// SIMATIC S7-200 project (STEP 7-Micro/WIN), CPU 226 REL 02.01

ORGANIZATION_BLOCK OB_1:OB1
TITLE=PROGRAM COMMENTS
// 食品或饮料行业的自动灌装机06 系统，通过启动灌装机，并在饮料瓶装生产线上精确控制瓶子的定位、灌装和封盖流程。
// 操作员按下启动按钮启动系统，设备通过上管控制将包装管送入位置，随后压板控制和压管控制分别在不同阶段固定管材。灌装阀和注料控制接着在各自脉冲范围内开始灌装液体。为了确保灌装一致性，注料控制和灌装阀应在编码器脉冲计数器的相同脉冲范围内动作，但目前两者的脉冲范围略有差异。运行状态指示灯在无故障信号A和故障信号B时点亮，显示设备运行，而启动按钮的信号通过其他逻辑参与控制。若故障信号A或故障信号B触发，例如电机故障或压力异常，运行状态指示灯立即熄灭。
// 系统通过编码器脉冲计数器精确记录灌装位置，色标传感器检测包装上的色标，确保灌装对准。灌装过程中，加热控制维持液体温度，但只有在冷却控制和风机控制均开启时才会激活，以避免温度失控。冷却控制、风机控制、搅拌控制和保温控制分别工作以维持灌装环境稳定，例如保持化妆品乳液的适宜粘度。若温度传感器检测到异常，系统暂停灌装并调整环境。压管传感器检测压管是否到位，置位压管到位标志，触发后续动作。
// 急停按钮被按下时，所有动作输出如上管控制、灌装阀、压板控制等应立即停止，但当前仅部分标志复位，需进一步完善。
BEGIN
Network 1
// 初始一次 on 系统初始化
LD     SM0.0
CALL   SBR_9:SBR9
?000
Network 2 // Network Title
// 运行初始化 （数据显示）
LD     SM0.1
CALL   SBR_0:SBR0
CALL   SBR_3:SBR3
=      M5.1
MOVW   +0, VW30
S      M1.1, 1
Network 3
// 恢复参数出厂设置
LD     M0.3
CALL   SBR_1:SBR1
Network 4
// 保存参数
LD     M0.4
CALL   SBR_2:SBR2
Network 5
// 参数修改后，未确定保存，参数恢复正常
LD     M2.4
CALL   SBR_3:SBR3
Network 6
// 大盘正常运行
LD     I1.2
O      M6.3
A      I0.5
AN     Q0.1
=      M6.3
EU
MOVW   +0, VW30
Network 7
// 点动运行
LD     I1.3
AN     Q0.1
=      M6.2
Network 8
LD     SM0.1
S      M2.0, 1
Network 9
// 大盘运行
LD     M6.2
O      M6.3
AN     Q0.1
EU
S      M20.6, 1
Network 10
// 点动停止
LD     M6.2
ED
R      M20.6, 1
Network 11
// 运行停机
LDD>=  HC0, +2300
AD<=   HC0, +2350
AN     M6.2
AN     M6.3
EU
R      M20.6, 1
Network 12
// 生产速度，计数设定，产量计数的BCD转换
LD     SM0.0
MOVW   VW10, VW54
BCDI   VW54
MOVW   VW14, VW50
BCDI   VW50
MOVW   VW52, VW18
IBCD   VW18
Network 13
// 手动升降速，及速度限制（速度必须在10-90之间)
LD     M1.1
LPS
AW>    VW54, +91
MOVW   +90, VW54
MOVW   VW54, VW10
IBCD   VW10
LRD
AW<    VW54, +10
MOVW   +10, VW54
MOVW   VW54, VW10
IBCD   VW10
LRD
AW<    VW54, +91
A      SM0.5
EU
A      M2.1
+I     +1, VW54
MOVW   VW54, VW10
IBCD   VW10
LPP
AW>    VW54, +10
A      SM0.5
EU
A      M2.2
-I     +1, VW54
MOVW   VW54, VW10
IBCD   VW10
Network 14
// 转速换算，根据大盘速度换算电机转速
LD     M1.1
MOVW   VW54, LW2
AENO
MUL    +44, LD0
AENO
MOVD   LD0, VD480
AENO
/D     +47, VD480
AENO
DTR    VD480, VD504
Network 15
// 真空 
LD     M1.1
A      M10.0
AN     M2.0
AN     Q0.1
=      Q0.7
Network 16
// 压板
LD     M1.1
AW>=   VW30, +2
A      M10.2
AN     M2.0
AN     M4.2
AD>=   HC0, VD140
AD<=   HC0, VD128
=      Q1.2
Network 17
// 上管
LD     M1.1
AW>=   VW30, +2
A      M2.7
AN     M2.0
AD>=   HC0, VD100
AD<=   HC0, +200
AN     M4.2
EU
S      Q0.2, 1
Network 18
// 上管回
LDD>=  HC0, +1150
ON     I0.5
EU
R      Q0.2, 1
Network 19
// 拨管
LD     M1.1
A      M10.2
AN     M2.0
AN     M4.2
=      Q1.3
Network 20
// 压管下
LD     M1.0
AW>=   VW30, +2
LD     M1.1
A      M10.1
OLD
AD>=   HC0, +1100
EU
S      Q1.7, 1
Network 21
// 净化，洗尘
LD     M3.0
A      M1.1
AD>=   HC0, VD104
AD<=   HC0, VD304
AN     M2.0
=      Q0.3
Network 22
// 停机复位 Q2.3未用 Q1.2压板 Q1.7压管 Q1.1灌装阀
LDN    M20.6
O      Q0.1
S      Q2.3, 1
R      Q1.2, 1
R      Q1.7, 1
EU
R      Q1.1, 1
Network 23
// 压管回
LD     I1.5
EU
R      Q1.7, 1
Network 24
// 允许脉冲输出,步进电机转动进行色标检测. M29.6状态取反（复位表示置位）
LDD>=  HC0, +1000
AD<=   HC0, +1050
EU
R      M29.6, 1
Network 25
// 禁止进行色标检测 M29.6状态取反（置位表示复位）
LDD>=  HC0, +1800
AD<=   HC0, +1850
EU
S      M29.6, 1
Network 26
// 色标电机停止转动 表示同步电机机械定位分开脱离停止旋转（上升结合旋转）
LDD>=  HC0, +2000
AD<=   HC0, +2050
MOVB   16#5, SMB67
PLS    0
Network 27
// 找到色标,步进停止转动
LD     I0.3
A      M20.5
LDN    I0.3
AN     M20.5
OLD
EU
MOVB   16#5, SMB67
PLS    0
Network 28
// 色标检测脉冲输出
LD     M1.1
A      M3.1
LDN    M25.0
A      I0.3
LD     M25.0
AN     I0.3
OLD
ALD
AN     M29.6
EU
AN     Q0.1
MOVB   16#85, SMB67
MOVW   +860, SMW68
MOVD   +99999999, SMD72
PLS    0
Network 29
// 检管信号记忆，注料启动
LDN    M2.0
ANI    I0.6
EU
S      M4.0, 1
Network 30
// 料塞
LD     M3.2
A      M1.1
AD>=   HC0, VD124
AD<=   HC0, VD132
AN     M2.0
A      M5.0
=      Q1.1
Network 31
// 注料
LD     M3.2
A      M1.1
AD>=   HC0, VD108
AD<=   HC0, VD112
AN     M2.0
A      M5.0
=      Q0.4
Network 32
// 吹气，并复位检管信号
LD     M3.2
A      M1.1
AD>=   HC0, VD116
AD<=   HC0, VD120
AN     M2.0
A      M5.0
=      Q0.5
Network 33
// 加热（必须先打开冷却，和风机才能正常工作）
LD     M1.0
O      M1.1
A      M10.4
A      Q1.6
A      Q1.5
=      Q1.4
NOT
R      M10.4, 1
Network 34
// 冷却
LD     M1.1
A      M10.3
O      Q1.5
=      Q1.5
Network 35
// 关闭冷却
LD     M10.3
ED
LPS
AN     M10.4
R      Q1.5, 1
LPP
A      M10.4
S      M10.3, 1
Network 36
// 风机
LD     M1.1
A      M3.3
O      Q1.6
=      Q1.6
Network 37
// 关闭风机
LD     M3.3
ED
LPS
AN     M10.4
R      Q1.6, 1
LPP
A      M10.4
S      M3.3, 1
Network 38
// 搅拌
LD     M1.1
A      M3.5
=      Q0.6
Network 39
// 保温
LD     M1.1
A      M3.6
=      Q1.0
Network 40
// 大盘运行停止,上管压管终止
LDN    M6.3
EU
R      M2.7, 1
R      M10.1, 2
Network 41
// 计数到标志位
LD     M1.4
AW>=   VW52, VW50
=      M4.2
Network 42
// 记数
LD     M1.1
AW<    VW52, VW50
A      Q0.4
EU
A      M1.4
INCW   VW52
Network 43
// 计数清零
LD     M1.3
MOVW   +0, VW52
Network 44
// 故障时，复位脉冲输出停机
LD     Q0.1
EU
R      M20.6, 1
MOVB   16#5, SMB67
PLS    0
Network 45
// USS协议
LD     SM0.0
=      L60.0
LD     M20.6
=      L63.7
LD     SM0.1
=      L63.6
LD     SM0.1
=      L63.5
LD     SM0.1
=      L63.4
LDN    SM0.0
=      L63.3
LD     L60.0
CALL   USS_CTRL:SBR8, L63.7, L63.6, L63.5, L63.4, L63.3, 1, 1, VD504, V500.3, VB514, VW516, VD510, V500.4, V500.5, V500.6, V500.7
Network 46
// 故障输出
LDN    I0.7
ON     I1.0
O      M13.0
=      Q0.1
Network 47
// 故障分类，触摸屏显示故障信息
LD     SM0.0
LPS
AN     I0.7
=      M20.0
LRD
AN     I1.0
=      M20.1
LPP
A      M13.0
=      M20.3
Network 48
// A门B门手盘车
LD     SM0.0
LPS
AN     I1.6
=      M13.1
LRD
AN     I1.7
=      M13.2
LPP
AN     I2.1
=      M13.3
Network 49
// 故障汇总
LD     M13.1
O      M13.3
O      M13.2
=      M13.0
Network 50
// 故障报警弹画面
LD     SM0.0
LPS
A      Q0.1
MOVW   +17, VW254
LPP
AN     Q0.1
EU
MOVW   +12, VW254
Network 51
// 画面值进行BCD转换
LD     SM0.0
MOVW   VW254, VW256
IBCD   VW256
Network 52
LD     SM0.0
DTI    HC0, VW180
MOVW   VW180, VW184
IBCD   VW184
END_ORGANIZATION_BLOCK

SUBROUTINE_BLOCK SBR_0:SBR0
TITLE=SUBROUTINE COMMENTS
BEGIN
Network 1 // Network Title
// Network Comment 开机时，所有数据清零
LD     SM0.0
R      Q0.0, 24
R      M0.0, 100
R      M10.0, 6
R      M25.0, 1
MOVD   +2330, VD1012
Network 2
// 高速计数器（编码器定义）
LD     SM0.0
MOVB   16#F8, SMB37
HDEF   0, 10
MOVD   +0, SMD38
MOVD   +30000, SMD42
ATCH   INT_0:INT0, 28
ENI
HSC    0
Network 3
// 步进电机脉冲定义（16#85为脉冲时间定义） SMD67脉冲参数 SMD68脉冲周期 SMD72脉冲数 (ATCH为中断控制  其中 INT_4 控制色标 7 为下降沿脉冲， 6 为上升沿脉冲)
LD     SM0.0
LPS
MOVB   16#85, SMB67
MOVW   +900, SMW68
MOVD   +99999999, SMD72
AN     M25.0
ATCH   INT_4:INT4, 7
LRD
A      M25.0
ATCH   INT_4:INT4, 6
LPP
ENI
Network 4
// 下列表示变频器与PLC之间通讯协议，1为模式 ，19200 为通讯速率， 16#02 为变频器地址 ， v500.0为变频器状态反馈地址（回答）
//  vb514为故障反馈地址
LD     SM0.0
CALL   USS_INIT:SBR5, 1, 19200, 16#2, V500.0, VB514
END_SUBROUTINE_BLOCK

SUBROUTINE_BLOCK SBR_1:SBR1
TITLE=
BEGIN
Network 1
// 机器工位编码器的脉冲位置（初始化时，将下列各值强制输入到设备内部）
LD     SM0.0
MOVW   +50, VW200
MOVW   +700, VW1004
MOVW   +800, VW208
MOVW   +1700, VW212
MOVW   +2000, VW216
MOVW   +2100, VW220
MOVW   +780, VW224
MOVW   +800, VW228
MOVW   +1600, VW232
MOVW   +2000, VW236
MOVW   +300, VW240
MOVW   +1800, VW150
Network 2
// 工位脉冲数值转换触摸屏代码显示
LD     SM0.0
MOVW   VW200, VW400
IBCD   VW400
MOVW   VW1004, VW404
IBCD   VW404
MOVW   VW208, VW408
IBCD   VW408
MOVW   VW212, VW412
IBCD   VW412
MOVW   VW216, VW416
IBCD   VW416
MOVW   VW220, VW420
IBCD   VW420
MOVW   VW224, VW424
IBCD   VW424
MOVW   VW228, VW428
IBCD   VW428
MOVW   VW232, VW432
IBCD   VW432
MOVW   VW236, VW436
IBCD   VW436
MOVW   VW240, VW440
IBCD   VW440
MOVW   VW150, VW152
IBCD   VW152
END_SUBROUTINE_BLOCK

SUBROUTINE_BLOCK SBR_2:SBR2
TITLE=
BEGIN
Network 1
// 确定数据保存（数据修改后确认）触摸屏及plc数据转换
LD     SM0.0
MOVW   VW400, VW200
BCDI   VW200
MOVW   VW404, VW1004
BCDI   VW1004
MOVW   VW408, VW208
BCDI   VW208
MOVW   VW412, VW212
BCDI   VW212
MOVW   VW416, VW216
BCDI   VW216
MOVW   VW420, VW220
BCDI   VW220
MOVW   VW424, VW224
BCDI   VW224
MOVW   VW428, VW228
BCDI   VW228
MOVW   VW432, VW232
BCDI   VW232
MOVW   VW436, VW236
BCDI   VW236
MOVW   VW440, VW240
BCDI   VW240
MOVW   VW152, VW150
BCDI   VW150
Network 2
LD     SM0.0
ITD    VW200, VD100
ITD    VW1004, VD104
ITD    VW208, VD108
ITD    VW212, VD112
ITD    VW216, VD116
ITD    VW220, VD120
ITD    VW224, VD124
ITD    VW228, VD128
ITD    VW232, VD132
ITD    VW236, VD136
ITD    VW240, VD140
ITD    VW150, VD160
Network 3
LD     SM0.0
MOVD   VD104, VD304
+D     +320, VD304
MOVD   VD128, VD328
+D     +256, VD328
END_SUBROUTINE_BLOCK

SUBROUTINE_BLOCK SBR_3:SBR3
TITLE=
BEGIN
Network 1
// 参数修改后，未确定保存，参数恢复未改动时状态
LD     SM0.0
DTI    VD100, VW200
DTI    VD104, VW1004
DTI    VD108, VW208
DTI    VD112, VW212
DTI    VD116, VW216
DTI    VD120, VW220
DTI    VD124, VW224
DTI    VD128, VW228
DTI    VD132, VW232
DTI    VD140, VW240
DTI    VD136, VW236
DTI    VD160, VW150
Network 2
LD     SM0.0
MOVW   VW200, VW400
IBCD   VW400
MOVW   VW1004, VW404
IBCD   VW404
MOVW   VW208, VW408
IBCD   VW408
MOVW   VW212, VW412
IBCD   VW412
MOVW   VW216, VW416
IBCD   VW416
MOVW   VW220, VW420
IBCD   VW420
MOVW   VW224, VW424
IBCD   VW424
MOVW   VW228, VW428
IBCD   VW428
MOVW   VW232, VW432
IBCD   VW432
MOVW   VW236, VW436
IBCD   VW436
MOVW   VW240, VW440
IBCD   VW440
MOVW   VW150, VW152
IBCD   VW152
Network 3
LD     SM0.0
R      M2.4, 1
END_SUBROUTINE_BLOCK

// SBR4: protected block, not included

// SBR5: protected block, not included

// SBR6: protected block, not included

// SBR7: protected block, not included

// SBR8: protected block, not included

SUBROUTINE_BLOCK SBR_9:SBR9
TITLE=子程序注释
BEGIN
Network 1
LD     SM0.0
A      SM0.4
LD     C3
CTU    C3, +60
Network 2
LD     SM0.0
A      C3
LD     C4
CTU    C4, +24
Network 3
LD     C4
EU
INCW   VW170
Network 4
LDW=   VW624, +30
LPS
EU
INCW   VW172
LPP
MOVW   +0, VW624
Network 5
LDW=   VW622, +12
LPS
EU
INCW   VW174
LPP
MOVW   +0, VW172
Network 6
LD     SM0.0
A      M14.0
EU
MOVW   +0, C3
MOVW   +0, C4
MOVW   +0, VW170
MOVW   +0, VW172
MOVW   +0, VW174
Network 7
LD     SM0.0
MOVW   C3, VW80
MOVW   C4, VW82
END_SUBROUTINE_BLOCK

INTERRUPT_BLOCK INT_0:INT0
TITLE=INTERRUPT ROUTINE COMMENTS
BEGIN
Network 1 // Network Title
// Network Comment
LD     M2.0
R      M2.0, 1
R      M4.1, 1
Network 2
LD     M1.1
AW<=   VW30, +29999
INCW   VW30
Network 3
LD     SM0.0
LPS
A      M4.0
S      M5.0, 1
LRD
AN     M4.0
R      M5.0, 1
LPP
R      M4.0, 1
Network 4
LD     SM0.0
CRETI
END_INTERRUPT_BLOCK

// INT1: protected block, not included

// INT2: protected block, not included

// INT3: protected block, not included

INTERRUPT_BLOCK INT_4:INT4
TITLE=
BEGIN
Network 1
LD     SM0.0
MOVB   16#5, SMB67
PLS    0
S      M29.6, 1
CRETI
END_INTERRUPT_BLOCK
